// Mitsubishi GX Works2 project: FXPLC_Client_1   PLC: FX3U/FX3UC
// FXPLC_Client_1

PROGRAM MAIN
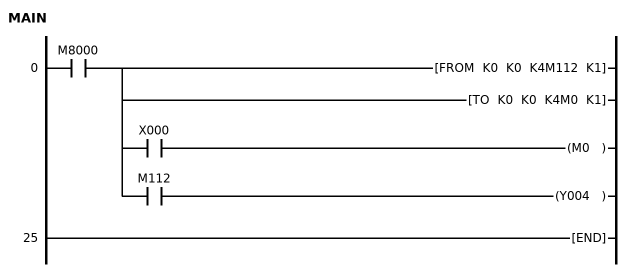
0     LD      M8000
      FROM    K0 K0 K4M112 K1
      TO      K0 K0 K4M0 K1
      MPS
      AND     X000
      OUT     M0
      MPP
      AND     M112
      OUT     Y004
25    END
END_PROGRAM
